(* Logix 5000 project; controller Transcat_L33ER vendor 1 type 14 code 107 rev 32.11; software revision 32.02; part 3 of 3 *)
(* tags used below, declared in another part *)
   alwaysOFF : BOOL;
   AnyAutoRun : BOOL;   // Bit that in on if ANY device is placed into Auto run (to signal pre-start beed)
   AnyManualRun : BOOL;   // Bit that in on if ANY device is placed into manual run (to signal pre-start beed)
   BeaconBlueLight : ALIAS FOR TC_Remote_IO:3:O.3;   // Blue Beacon Light
   BeaconGreenLight : ALIAS FOR TC_Remote_IO:3:O.2;   // Green Beacon Light
   BeaconRedLight : ALIAS FOR TC_Remote_IO:3:O.0;   // Red Beacon Light
   BeaconYellowLight : ALIAS FOR TC_Remote_IO:3:O.1;   // Yellow Beacon Light
   Beep : BOOL;   // Bit to Activte Beacon Alarm
   BeepNew : ALIAS FOR TC_Remote_IO:3:O.4;
   FT103 : BronkhorstFlowMeter;
   FT104 : BronkhorstFlowMeter;
   FT105 : BronkhorstFlowMeter;
   GF101 : Thayer_WB_Feeder;   // Thayer 1 Tags
   GF201 : Thayer_WB_Feeder;   // Thayer 2 Tags
   GF301 : Acrison_Feeder;   // GF103 - Small Feeder 1
   GreenFlashingOff : TIMER;
   GreenFlashingOn : TIMER;
   MSG_FROM_SLC500 : INT[10];
   MX101 : Howes_Mixer;
   MX201 : Howes_Mixer;
   StartBeepTimer : TIMER;   // Timer to sound the beep alarm before starting a device
   UpperHowesSpeed : INT;
   VF101 : Acrison_Feeder;   // Medium Feeder Tags
   VF201 : Acrison_Feeder;   // Small Feeder 2 Tags
   VFD_Panel_Safety_Hoist_1_Cart_OK : ALIAS FOR XS26_VFD_Cabinet_Safety_Controller:I1.Data[2].2;   // HOIST 1 Cart Sensor
   VFD_Panel_Safety_Hoist_2_Cart_OK : ALIAS FOR XS26_VFD_Cabinet_Safety_Controller:I1.Data[2].3;   // HOIST 2 Cart Sensor
   YellowFlashOff : TIMER;
   YellowFlashOn : TIMER;
(* MainProgram, continued *)

ROUTINE Light_Beacon   (* ladder *)
// Indicator Light Beacon
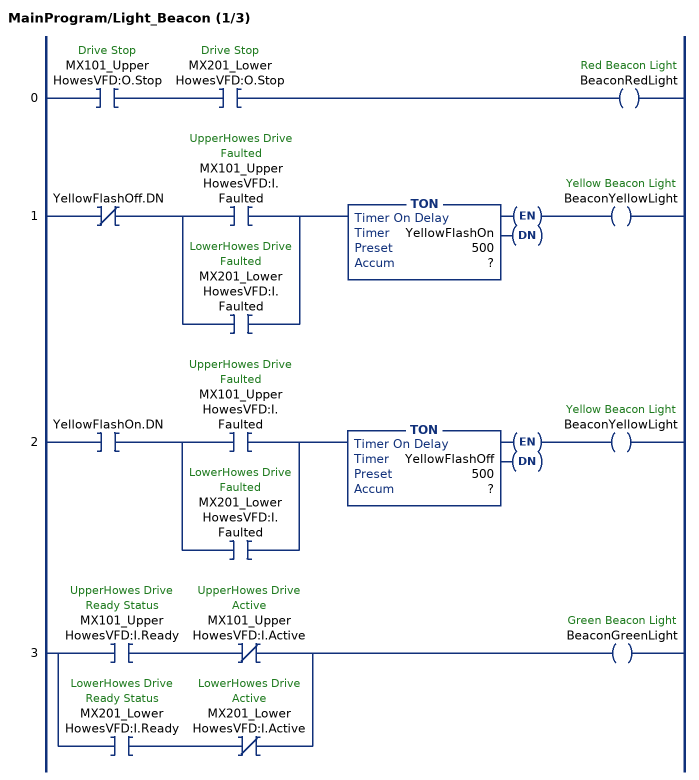
   0: XIC(MX101_UpperHowesVFD:O.Stop)XIC(MX201_LowerHowesVFD:O.Stop)OTE(BeaconRedLight);
   1: XIO(YellowFlashOff.DN)[XIC(MX101_UpperHowesVFD:I.Faulted) ,XIC(MX201_LowerHowesVFD:I.Faulted) ]TON(YellowFlashOn,?,?)OTE(BeaconYellowLight);
   2: XIC(YellowFlashOn.DN)[XIC(MX101_UpperHowesVFD:I.Faulted) ,XIC(MX201_LowerHowesVFD:I.Faulted) ]TON(YellowFlashOff,?,?)OTE(BeaconYellowLight);
   3: [XIC(MX101_UpperHowesVFD:I.Ready) XIO(MX101_UpperHowesVFD:I.Active) ,XIC(MX201_LowerHowesVFD:I.Ready) XIO(MX201_LowerHowesVFD:I.Active) ]OTE(BeaconGreenLight);
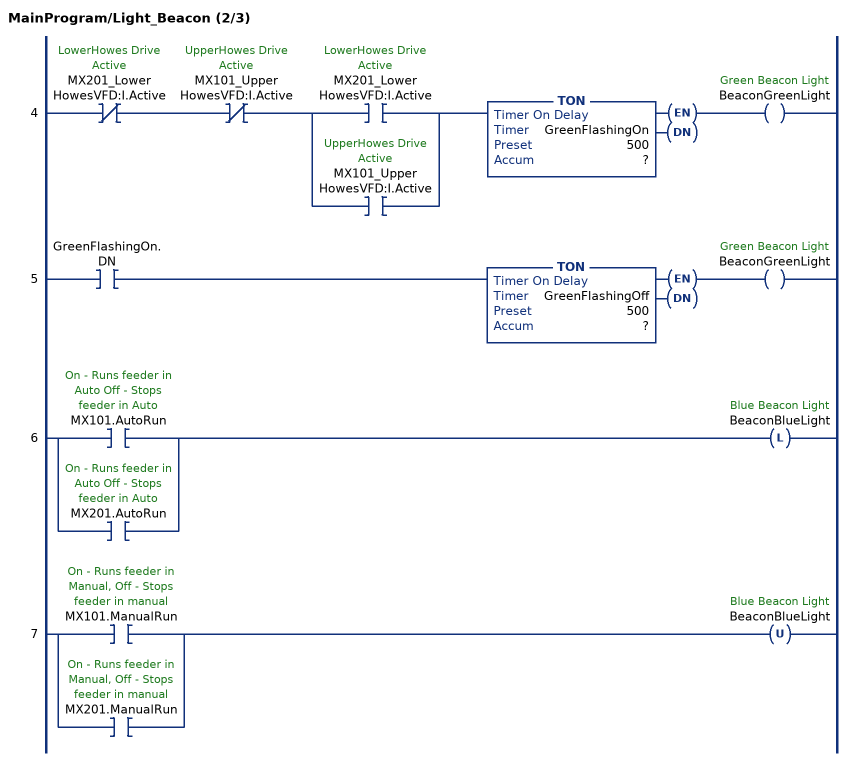
   4: XIO(MX201_LowerHowesVFD:I.Active)XIO(MX101_UpperHowesVFD:I.Active)[XIC(MX201_LowerHowesVFD:I.Active) ,XIC(MX101_UpperHowesVFD:I.Active) ]TON(GreenFlashingOn,?,?)OTE(BeaconGreenLight);
   5: XIC(GreenFlashingOn.DN)TON(GreenFlashingOff,?,?)OTE(BeaconGreenLight);
   6: [XIC(MX101.AutoRun) ,XIC(MX201.AutoRun) ]OTL(BeaconBlueLight);
   7: [XIC(MX101.ManualRun) ,XIC(MX201.ManualRun) ]OTU(BeaconBlueLight);
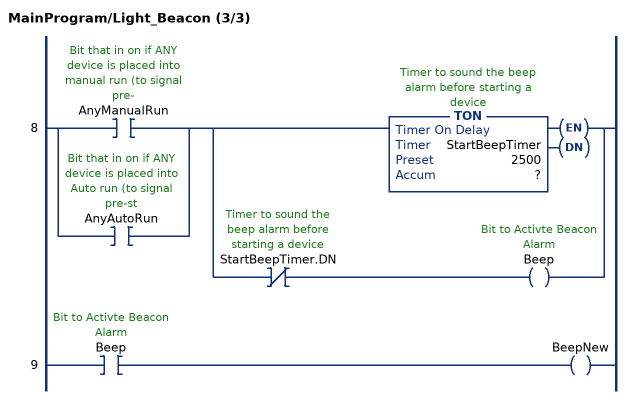
   8: [XIC(AnyManualRun) ,XIC(AnyAutoRun) ][TON(StartBeepTimer,?,?) ,XIO(StartBeepTimer.DN) OTE(Beep) ];
   9: XIC(Beep)OTE(BeepNew);
END_ROUTINE

ROUTINE MainRoutine   (* ladder *)
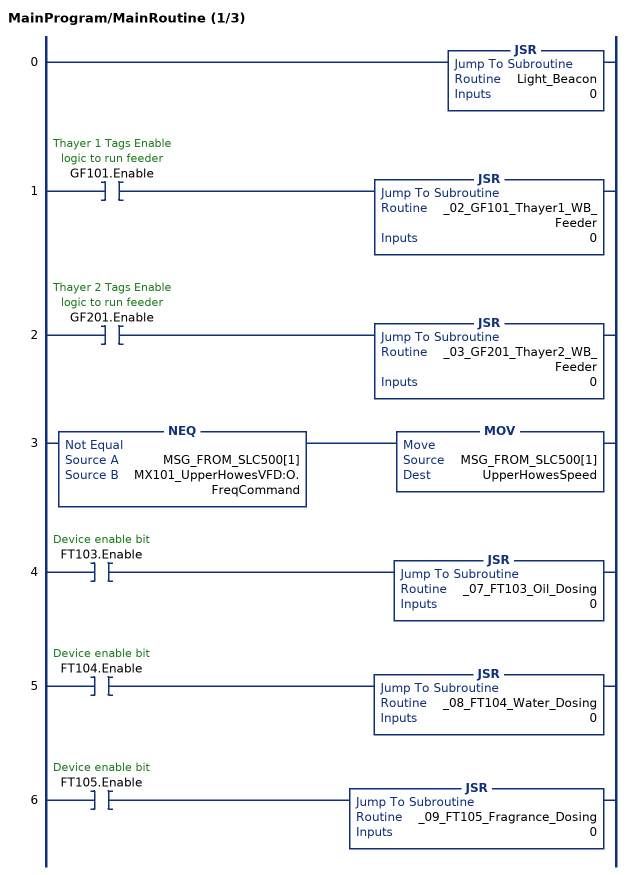
   0: JSR(Light_Beacon,0);
   1: XIC(GF101.Enable)JSR(_02_GF101_Thayer1_WB_Feeder,0);
   2: XIC(GF201.Enable)JSR(_03_GF201_Thayer2_WB_Feeder,0);
   3: NEQ(MSG_FROM_SLC500[1],MX101_UpperHowesVFD:O.FreqCommand)MOV(MSG_FROM_SLC500[1],UpperHowesSpeed);
   4: XIC(FT103.Enable)JSR(_07_FT103_Oil_Dosing,0);
   5: XIC(FT104.Enable)JSR(_08_FT104_Water_Dosing,0);
   6: XIC(FT105.Enable)JSR(_09_FT105_Fragrance_Dosing,0);
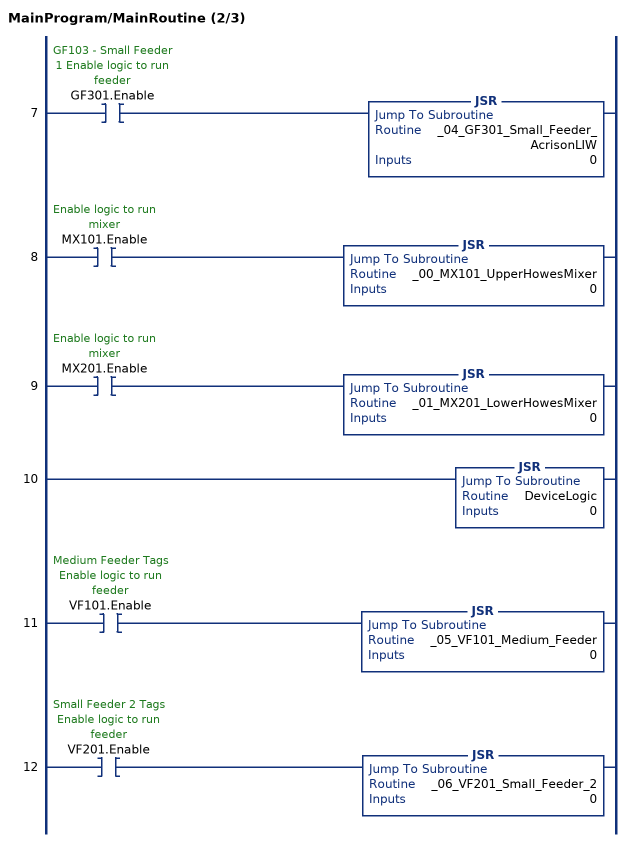
   7: XIC(GF301.Enable)JSR(_04_GF301_Small_Feeder_AcrisonLIW,0);
   8: XIC(MX101.Enable)JSR(_00_MX101_UpperHowesMixer,0);
   9: XIC(MX201.Enable)JSR(_01_MX201_LowerHowesMixer,0);
   10: JSR(DeviceLogic,0);
   11: XIC(VF101.Enable)JSR(_05_VF101_Medium_Feeder,0);
   12: XIC(VF201.Enable)JSR(_06_VF201_Small_Feeder_2,0);
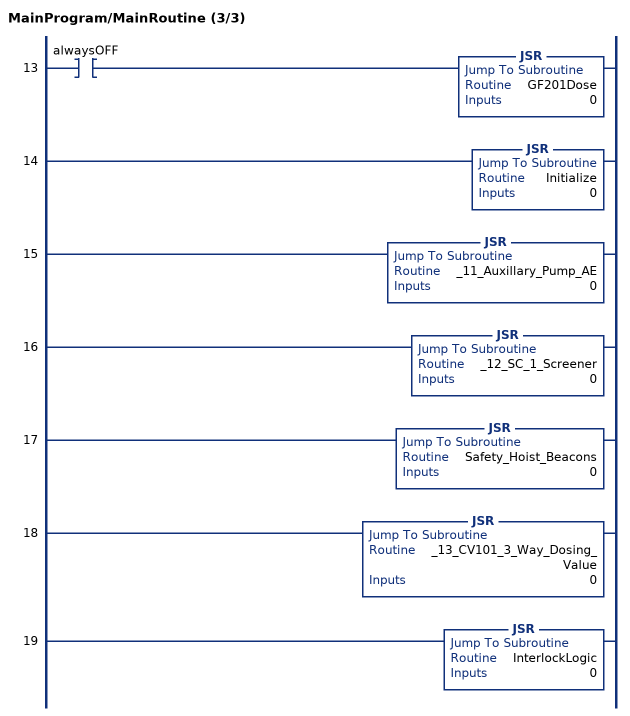
   13: XIC(alwaysOFF)JSR(GF201Dose,0);
   14: JSR(Initialize,0);
   15: JSR(_11_Auxillary_Pump_AE,0);
   16: JSR(_12_SC_1_Screener,0);
   17: JSR(Safety_Hoist_Beacons,0);
   18: JSR(_13_CV101_3_Way_Dosing_Value,0);
   19: JSR(InterlockLogic,0);
END_ROUTINE

ROUTINE Safety_Hoist_Beacons   (* ladder *)
// Saety Hoist Light Beacons
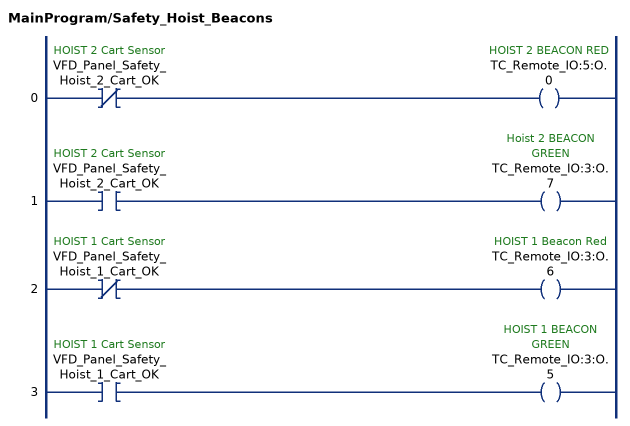
   0: XIO(VFD_Panel_Safety_Hoist_2_Cart_OK)OTE(TC_Remote_IO:5:O.0);
   1: XIC(VFD_Panel_Safety_Hoist_2_Cart_OK)OTE(TC_Remote_IO:3:O.7);
   2: XIO(VFD_Panel_Safety_Hoist_1_Cart_OK)OTE(TC_Remote_IO:3:O.6);
   3: XIC(VFD_Panel_Safety_Hoist_1_Cart_OK)OTE(TC_Remote_IO:3:O.5);
END_ROUTINE
END_PROGRAM
